RESOURCE_TYPE top
  (* Standard: 61499-2 *)
  (* Version 0.1, 2017-00-25, hpea485, UOA *)
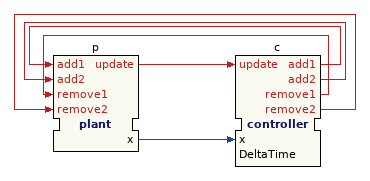
  FBS
    p : plant;
    c : controller;
  END_FBS
  EVENT_CONNECTIONS
    p.update TO c.update;
    c.add1 TO p.add1;
    c.add2 TO p.add2;
    c.remove1 TO p.remove1;
    c.remove2 TO p.remove2;
  END_CONNECTIONS
  DATA_CONNECTIONS
    p.x TO c.x;
  END_CONNECTIONS
END_RESOURCE_TYPE
